// TIA Portal V15.1 export
// export: Created 2026-01-09T13:45:11.8978607Z, ExportSetting WithDefaults, WithReadOnly, DisplayName Totally Integrated Automation Portal, DisplayVersion V15.1 Update 8, DisplayName TIA Portal Openness, DisplayVersion V15.1 Update 8, DisplayName STEP 7 Professional, DisplayVersion V15.1 Update 8, DisplayName WinCC Advanced, DisplayVersion V15.1 Update 8
DATA_BLOCK "PLC_DATA"   // DB10
{ S7_Optimized_Access := 'FALSE' }
VERSION : 0.1
// stored: AutoNumber true, CodeModifiedDate 2026-01-04T14:16:44.6751265Z, CompileDate 2026-01-04T14:27:04.9564115Z, CreationDate 2024-10-12T12:36:08.0193576Z, DBAccessibleFromOPCUA true, InterfaceModifiedDate 2026-01-04T14:16:44.6751265Z, IsConsistent true, IsKnowHowProtected false, IsOnlyStoredInLoadMemory false, IsPLCDB false, IsWriteProtectedInAS false, ModifiedDate 2026-01-04T14:16:44.6751265Z, ParameterModified 2026-01-04T14:16:44.6751265Z, StructureModified 2026-01-04T14:16:44.6751265Z
   VAR RETAIN
      SI_WAG : Real;
      RE_WAG : Real;
      SI_WFD : Real;
      RE_WFD : Real;
      SI_WAP : Real;
      RE_WAP : Real;
      SI_WSB : Real;
      RE_WSB : Real;
      TEMP_TL : DInt;
      TEMP_TS : DInt;
      TEMP_AG : DInt;
      TEMP_AP : DInt;
      TG_TRON : Real;
      TG_XA : Real;
      M3_MAX : Real;
      SMC_SILO_AG1 : Real;
      SMC_SILO_AG2 : Real;
      SMC_SILO_AG3 : Real;
      SMC_SILO_AG4 : Real;
      SMC_SILO_AG5 : Real;
      SMC_SILO_FD1 : Real;
      SMC_SILO_AP1 : Real;
      SMC_SILO_SB1 : Real;
      SI_WAGG1 : Real;
      RE_WAGG1 : Real;
      SI_WAGG2 : Real;
      RE_WAGG2 : Real;
      SI_WAGG3 : Real;
      RE_WAGG3 : Real;
      SI_WAGG4 : Real;
      RE_WAGG4 : Real;
      SI_WAGG5 : Real;
      RE_WAGG5 : Real;
   END_VAR
BEGIN
END_DATA_BLOCK
